VAR_GLOBAL PERSISTENT

	iZAxisUpperLimitValue: DINT;
	iZAxisLowerLimitValue: DINT;
	lTeachLimitRight: LREAL;
	lTeachLimitLeft: LREAL;
END_VAR

(* stored: Version 1.1.0.1, ProductVersion 3.1.4024.15
   GVL GVL_Persistent: Id {14440726-a52a-4e9b-b498-089c0f0ea337} *)
